{attribute 'qualified_only'}
{attribute 'strict'}
TYPE ProfileJerkSigns :
(
	Uddu,
  Udud 
);
END_TYPE

(* stored: Version 1.1.0.1
   DUT ProfileJerkSigns: Id {b8a5c43f-13de-4042-9633-9e96e9516e46} *)
